PROGRAM LogicalCircuits_Ex02
VAR
	S1					: WorkshopLibrary.DigitalInputNO;
	S2					: WorkshopLibrary.DigitalInputNO;
	P1					: WorkshopLibrary.DigitalOutput;
END_VAR

// Evaluate inputs
S1(input := GVL_IO.input01);
S2(input := GVL_IO.input02);

// process outputs
P1(on:=S1.isActive AND S2.isActive, output=>GVL_IO.output01);

END_PROGRAM

(* stored: Version 1.1.0.1
   POU LogicalCircuits_Ex02: Id {928081cd-c731-4064-9f20-4dd0f589a3e1}, SpecialFunc None *)
